(* PLC project Unnamed, Unknown Unnamed 1 *)
(* stored: creationDateTime 2025-02-21T14:25:40, modificationDateTime 2025-03-03T20:36:31 *)

PROGRAM Mixing
  VAR
    m AT %QX0.0 : BOOL;  (* Starting button *)
    a AT %QX0.1 : BOOL;  (* Position sensor placed on the valve A *)
    b AT %QX0.2 : BOOL;  (* Position sensor placed on the valve B *)
    d1 AT %QX0.3 : BOOL;  (* Weight sensor that controls the weight of the materials inside the valve D according to the fixed quantity *)
    d2 AT %QX0.4 : BOOL;  (* Position sensor placed on the valve D *)
    e1 AT %QX0.5 : BOOL;  (* Weight sensor that controls the weight of the materials inside the valve E according to the fixed quantity *)
    e2 AT %QX0.6 : BOOL;  (* Position sensor placed on the valve D *)
    f AT %QX0.7 : BOOL;  (* Position sensor placed in front of the motor M1 *)
    g AT %QX1.0 : BOOL;  (* Position sensor placed in front of the motor M2 *)
    l AT %QX1.1 : BOOL;  (* Sensor that measures the level of the liquid inside the pipe *)
    EA AT %QX2.0 : BOOL;  (* Cylinder controlling the opening and the closing of the valve A *)
    EB AT %QX2.1 : BOOL;  (* Cylinder controlling the opening and the closing of the valve B *)
    ED AT %QX2.2 : BOOL;  (* Cylinder controlling the opening and the closing of the valve C *)
    EE AT %QX2.3 : BOOL;  (* Cylinder controlling the opening and the closing of the valve D *)
    EF AT %QX2.4 : BOOL;  (* Cylinder controlling the opening and the closing of the valve attached to the engine M1 *)
    EG AT %QX2.5 : BOOL;  (* Cylinder controlling the opening and the closing of the vessel *)
    M1 AT %QX2.6 : BOOL;  (* 3D mixer engine *)
    M2 AT %QX2.7 : BOOL;  (* Inline-mixer (high shear) engine *)
    X0 AT %QX3.0 : BOOL := TRUE;  (* Step 0 *)
    X1 AT %QX3.1 : BOOL;  (* Step 1 *)
    X2 AT %QX3.2 : BOOL;  (* Step 2 *)
    X3 AT %QX3.3 : BOOL;  (* Step 3 *)
    X4 AT %QX3.4 : BOOL;  (* Step 4 *)
    X5 AT %QX3.5 : BOOL;  (* Step 5 *)
    X6 AT %QX3.6 : BOOL;  (* Step 6 *)
    X7 AT %QX3.7 : BOOL;  (* Step 7 *)
    X8 AT %QX4.0 : BOOL;  (* Step 8 *)
    T0 AT %QX5.0 : BOOL;  (* Transition 0 *)
    T1 AT %QX5.1 : BOOL;  (* Transition 1 *)
    T2 AT %QX5.2 : BOOL;  (* Transition 2 *)
    T3 AT %QX5.3 : BOOL;  (* Transition 3 *)
    T4 AT %QX5.4 : BOOL;  (* Transition 4 *)
    T5 AT %QX5.5 : BOOL;  (* Transition 5 *)
    T6 AT %QX5.6 : BOOL := FALSE;  (* Transition 6 *)
    T7 AT %QX5.7 : BOOL := FALSE;  (* Transition 7 *)
    T8 AT %QX6.0 : BOOL := FALSE;  (* Transition 8 *)
    PV AT %QW0 : INT := 3;  (* Preset Value *)
    CV AT %QW1 : INT;  (* Counting Value *)
    time_1 AT %QW2 : INT := 0;  (* Timer 1 *)
    time_2 AT %QW3 : INT := 0;  (* Timer 2 *)
    timer_gauge_1 AT %QW4 : INT := 5;  (* Timer button of the engine M1 *)
    timer_gauge_2 AT %QW5 : INT := 5;  (* Timer button of the 3D mixer M1 *)
    CU AT %QX7.0 : BOOL := TRUE;  (* Counting Unit *)
  END_VAR
  VAR
    TP1 : TP;
    TP2 : TP;
    CTU0 : CTU;
    TON0 : TON;
  END_VAR
  VAR  (* added by the conversion: wires and edge detectors of the diagram *)
    R_TRIG1 : R_TRIG;
  END_VAR

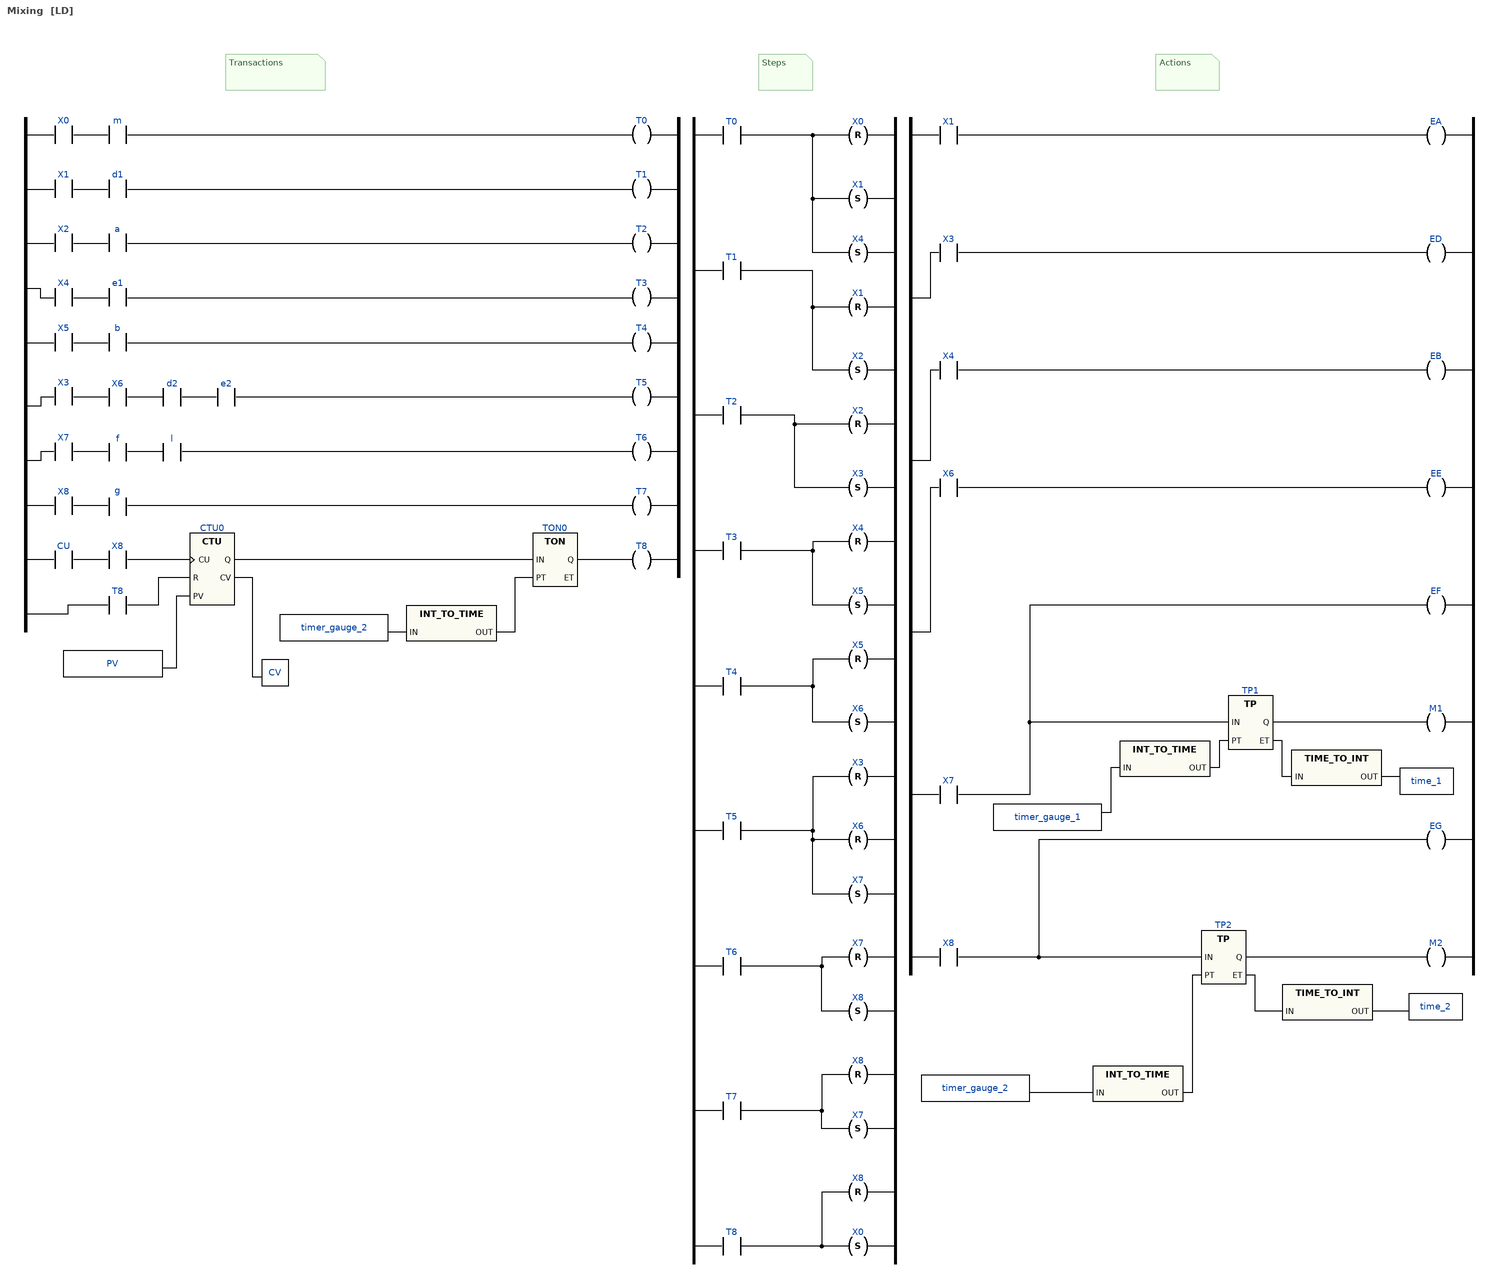
(* LD diagram, written out as Structured Text *)
(* Transactions *)
(* Steps *)
(* Actions *)
T0 := X0 AND m;
T1 := X1 AND d1;
T2 := X2 AND a;
T3 := X4 AND e1;
T4 := X5 AND b;
T5 := X3 AND X6 AND d2 AND e2;
IF T0 THEN X0 := FALSE; END_IF;
IF T0 THEN X1 := TRUE; END_IF;
IF T0 THEN X4 := TRUE; END_IF;
IF T1 THEN X1 := FALSE; END_IF;
IF T1 THEN X2 := TRUE; END_IF;
IF T2 THEN X2 := FALSE; END_IF;
IF T2 THEN X3 := TRUE; END_IF;
IF T3 THEN X4 := FALSE; END_IF;
IF T3 THEN X5 := TRUE; END_IF;
IF T4 THEN X5 := FALSE; END_IF;
IF T4 THEN X6 := TRUE; END_IF;
IF T5 THEN X3 := FALSE; END_IF;
IF T5 THEN X6 := FALSE; END_IF;
IF T6 THEN X7 := FALSE; END_IF;
IF T6 THEN X8 := TRUE; END_IF;
EA := X1;
ED := X3;
EB := X4;
EE := X6;
EF := X7;
TP2(IN := X8, PT := INT_TO_TIME(timer_gauge_2));
M2 := TP2.Q;
TP1(IN := X7, PT := INT_TO_TIME(timer_gauge_1));
M1 := TP1.Q;
EG := X8;
R_TRIG1(CLK := CU AND X8);
CTU0(CU := R_TRIG1.Q, R := T8, PV := PV);
TON0(IN := CTU0.Q, PT := INT_TO_TIME(timer_gauge_2));
T8 := TON0.Q;
CV := CTU0.CV;
T6 := X7 AND f AND l;
IF T5 THEN X7 := TRUE; END_IF;
IF T7 THEN X8 := FALSE; END_IF;
IF T7 THEN X7 := TRUE; END_IF;
IF T8 THEN X8 := FALSE; END_IF;
IF T8 THEN X0 := TRUE; END_IF;
T7 := X8 AND g;
time_1 := TIME_TO_INT(TP1.ET);
time_2 := TIME_TO_INT(TP2.ET);
END_PROGRAM

CONFIGURATION Config0
  RESOURCE Res0 ON PLC
    TASK task0(INTERVAL := T#20ms, PRIORITY := 0);
    PROGRAM instance0 WITH task0 : Mixing;
  END_RESOURCE
END_CONFIGURATION
